// TIA Portal V15.1 export
// export: Created 2026-01-09T13:45:11.8030122Z, ExportSetting WithDefaults, WithReadOnly, DisplayName Totally Integrated Automation Portal, DisplayVersion V15.1 Update 8, DisplayName TIA Portal Openness, DisplayVersion V15.1 Update 8, DisplayName STEP 7 Professional, DisplayVersion V15.1 Update 8, DisplayName WinCC Advanced, DisplayVersion V15.1 Update 8
DATA_BLOCK "C#7_RD_RUN"   // DB7
{ S7_Optimized_Access := 'FALSE' }
VERSION : 0.1
// stored: AutoNumber true, CodeModifiedDate 2024-10-13T07:13:35.9743236Z, CompileDate 2025-08-30T17:40:32.1468413Z, CreationDate 2024-10-12T12:36:08.0193576Z, DBAccessibleFromOPCUA true, InterfaceModifiedDate 2024-10-13T07:13:35.9743236Z, IsConsistent true, IsKnowHowProtected false, IsOnlyStoredInLoadMemory false, IsPLCDB false, IsWriteProtectedInAS false, ModifiedDate 2024-10-13T07:14:11.4381467Z, ParameterModified 2024-10-13T07:13:35.9743236Z, StructureModified 2024-10-13T07:13:35.9743236Z
   VAR RETAIN
      PV_AG1 : Real;   // Thực cân cốt liệu 1
      "%_WAG1" : Real;   // Phần trăm khối lượng cốt liệu 1
      WE_AG1 : Real;   // Khối lượng cân cốt liệu 1
      SMC_AG1 : Real;   // Số mẻ cân phễu cân cốt liệu 1
      SMX_AG1 : Real;   // Số mẻ xả phễu cân cốt liệu 1
      PV_AG2 : Real;   // Thực cân cốt liệu 2
      SMC_AG2 : Real;   // Số mẻ cân phễu cân cốt liệu 2
      SMX_AG2 : Real;   // Số mẻ xả phễu cân cốt liệu 2
      PV_AG3 : Real;   // Thực cân cốt liệu 3
      SMC_AG3 : Real;   // Số mẻ cân phễu cân cốt liệu 3
      SMX_AG3 : Real;   // Số mẻ xả phễu cân cốt liệu 3
      PV_AG4 : Real;   // Thực cân cốt liệu 4
      SMC_AG4 : Real;   // Số mẻ cân phễu cân cốt liệu 4
      SMX_AG4 : Real;   // Số mẻ xả phễu cân cốt liệu 4
      PV_AG5 : Real;   // Thực cân cốt liệu 5
      SMC_AG5 : Real;   // Số mẻ cân phễu cân cốt liệu 5
      SMX_AG5 : Real;   // Số mẻ xả phễu cân cốt liệu 5
      PV_FD1 : Real;   // Thực cân silo FD 1
      "%_WFD1" : Real;   // Phần trăm khối lượng phễu cân FD 1
      WE_FD1 : Real;   // Khối lượng phễu cân FD 1
      SMC_FD1 : Real;   // Số mẻ cân phễu cân FD 1
      SMX_FD1 : Real;   // Số mẻ xả phễu cân FD 1
      PV_AP1 : Real;   // Thực cân Nhựa 1
      "%_WAP1" : Real;   // Phần trăm khối lượng phễu cân Nhựa 1
      WE_AP1 : Real;   // Khối lượng phễu cân Nhựa 1
      SMC_AP1 : Real;   // Số mẻ cân phễu cân Nhựa 1
      SMX_AP1 : Real;   // Số mẻ xả phễu cân Nhựa 1
      PV_SB1 : Real;   // Thực cân SBS 1
      "%_WSB1" : Real;   // Phần trăm khối lượng phễu cân SBS 1
      WE_SB1 : Real;   // Khối lượng phễu cân SBS 1
      SMC_SB1 : Real;   // Số mẻ cân phễu cân SBS 1
      SMX_SB1 : Real;   // Số mẻ xả phễu cân SBS 1
      SMC_MIXER : Real;   // Số mẻ cân nồi trộn
      SMX_MIXER : Real;   // Số mẻ xả nồi trộn
      "TG_THUC TRON" : Real;   // Thoi gian thuc tron
      TG_THUC_XA : Real;   // Thoi gian thuc xa
      SMT : Real;
      "M3/ME" : Real;
      PVM_AG1 : Real;   // Thực cân tay cốt liệu 1
      PVM_AG2 : Real;   // Thực cân tay cốt liệu 2
      PVM_AG3 : Real;   // Thực cân tay cốt liệu 3
      PVM_AG4 : Real;   // Thực cân tay cốt liệu 4
      PVM_AG5 : Real;   // Thực cân tay cốt liệu 5
      PVM_FD1 : Real;   // Thực cân tay FD1
      PVM_AP1 : Real;   // Thực cân tay Nhựa
      PVM_SB1 : Real;   // Thực cân tay SBS1
      TEMP_TUILOC : Real;   // Nhiệt độ túi lọc hiển thị
      TEMP_AGG : Real;   // Nhiệt độ cốt liệu hiển thị
      TEMP_TANSAY : Real;   // Nhiệt độ tan sấy hiển thị
      TEMP_NHUA : Real;   // Nhiệt độ nhựa hiển thị
   END_VAR
BEGIN
END_DATA_BLOCK
